FUNCTION_BLOCK SSC_TransferWorkpieceTo_PSStart EXTENDS SSC_MoveWorkpiece_Base
VAR_INPUT
END_VAR
VAR_OUTPUT
END_VAR
VAR
	// (EProcessVariables.PicAlpha_HoldingWorkpiece = FALSE) AND ((EProcessVariables.PicAlpha_CylinderRetracted = TRUE) AND (EProcessVariables.PicAlpha_AtPos4 = TRUE))
	m_compExpr226: ComparisonExpression(EProcessVariables.PicAlpha_HoldingWorkpiece, EComparisonType.equals, EDataType.binary, FALSE, 0, '', TRUE);
	m_compExpr228: ComparisonExpression(EProcessVariables.PicAlpha_CylinderRetracted, EComparisonType.equals, EDataType.binary, TRUE, 0, '', TRUE);
	m_compExpr230: ComparisonExpression(EProcessVariables.PicAlpha_AtPos4, EComparisonType.equals, EDataType.binary, TRUE, 0, '', TRUE);
	m_boolExpr231: BoolExpression(m_compExpr228, EBoolOperation.and_op, m_compExpr230);
	m_precondition: BoolExpression(m_compExpr226, EBoolOperation.and_op, m_boolExpr231);
	
	// EProcessVariables.SSC_WPAtStart = TRUE
	m_postcondition: ComparisonExpression(EProcessVariables.SSC_WPAtStart, EComparisonType.equals, EDataType.binary, TRUE, 0, '', TRUE);
END_VAR

SUPER^();

METHOD PROTECTED  AtTarget : BOOL
VAR_INPUT
END_VAR
//AtTarget := FALSE;
IF m_ptrSSC^.WPAtStart THEN
	AtTarget := TRUE;
END_IF
END_METHOD

METHOD FB_init : BOOL
VAR_INPUT
	bInitRetains : BOOL; // if TRUE, the retain variables are initialized (warm start / cold start)
	bInCopyCode : BOOL;  // if TRUE, the instance afterwards gets moved into the copy code (online change)
	
	i_ptrSSC: POINTER TO SmallSortingConveyor;
END_VAR
m_ptrSSC := i_ptrSSC;

m_id := EPrimitives.SSC_TransferWorkpieceTo_PSStart;
m_timeout := T#200S;

Precondition := m_precondition;
Postcondition := m_postcondition;
END_METHOD

END_FUNCTION_BLOCK

(* stored: Version 1.1.0.1, ProductVersion 3.1.4024.9
   POU SSC_TransferWorkpieceTo_PSStart: Id {ee0b64a7-03b0-43b4-a161-102b62cf41f7}, SpecialFunc None
   Method AtTarget: Id {9c01a3dc-2f21-420a-a04b-77dc2ddbebee}
   Method FB_init: Id {17531b7f-ff49-436d-9003-99fab6e3e9d0} *)
